ABB RobotStudio station: project.rsstn

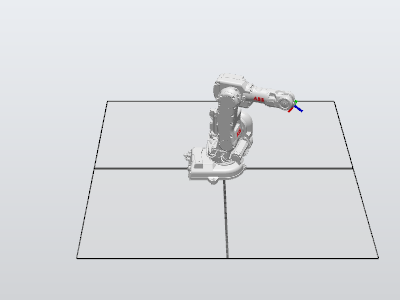
Station Station (saved by RobotStudio 22.3.10190.2)
Controller IRB140_6_81_1
  mechanical unit ROB_1: IRB140_6_81_C_03, 6 joints, base frame (0, 0, 0) mm
Layout (positions relative to the parent item):
  - IRB140_6_81_C_03 [mechanism, from Robots\IRB140_6_81_C_G_03.rslib] at (0, 0, 0) mm; joint values [-0.347, 0, 0, 0, 0.5236, 0] (rad or m)
